(* Schneider Machine Expert - Basic project Run Hour, file version 1.7.0.0 *)
(* ProjectInformations: Name=New project *)

HARDWARE
  Cpu 0: TM221ME32TK
  EthernetConfiguration: NetworkName=M221, IpAllocationMode=FixedAddress, IpAddress=0.0.0.0, SubnetMask=0.0.0.0
  SerialLineConfiguration: Baud=Baud19200, Parity=ParityEven, DataBits=DataBits8, StopBits=StopBits1, PhysicalMedium=PhysicalMediumRs485, TransmissionMode=TransmissionModeModbusRtu, SlaveId=1, Addressing=SlaveAddressing
  MastTask: UsePeriodScanMode=false, PeriodScan=100
  FastTask: Period=255
  CpuBehavior: StartingMode=StartAsPreviousState, AutoSaveRamOnEeprom=true, WatchdogPeriod=250

SYMBOLS  (address, symbol, comment, settings)
  %TM1        "T1"  [Preset=5, Base=OneSecond]
  %TM2        "T2"  [Preset=5, Base=OneSecond]
  %TM3        [Base=OneSecond, IsRetentive=true]
  %TM4        [Base=OneSecond, IsRetentive=true]
  %I0.0       "Auto"
  %I0.1       "Manual"
  %I0.2       "Pompa 1"
  %I0.3       "Pompa 2"
  %Q0.0       "P1"
  %Q0.1       "P2"

POU New POU
  (* SectionNumber=1 *)

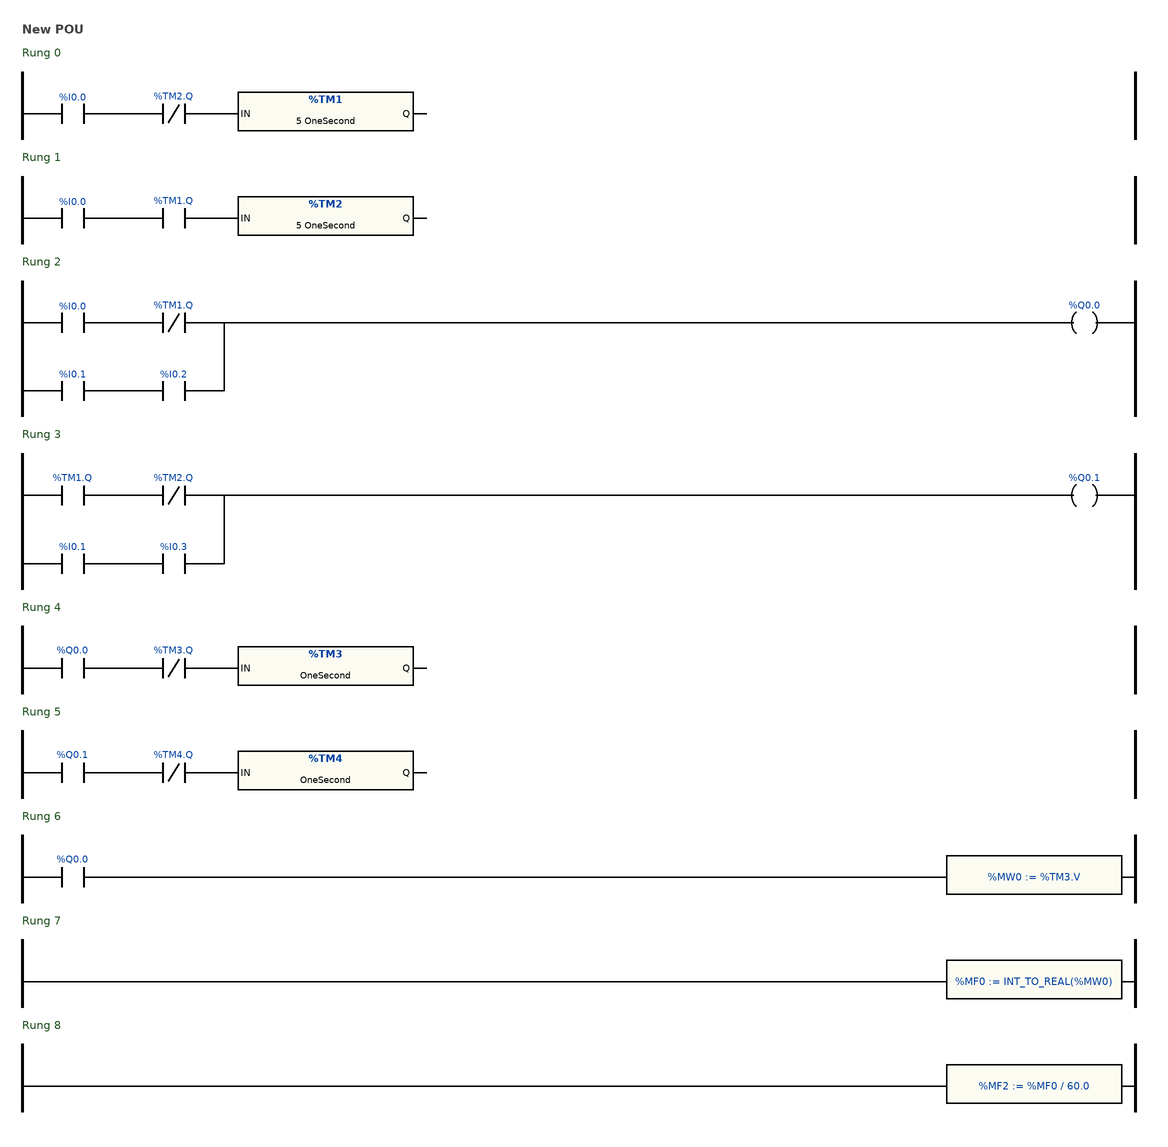

// Rung 0
  BLK %TM1
  LD %I0.0
  ANDN %TM2.Q
  IN
  END_BLK
  // as ST:
  //   %TM1(IN := %I0.0 AND NOT %TM2.Q);

// Rung 1
  BLK %TM2
  LD %I0.0
  AND %TM1.Q
  IN
  END_BLK
  // as ST:
  //   %TM2(IN := %I0.0 AND %TM1.Q);

// Rung 2
  LD %I0.0
  ANDN %TM1.Q
  OR( %I0.1
  AND %I0.2
  )
  ST %Q0.0
  // as ST:
  //   %Q0.0 := %I0.0 AND NOT %TM1.Q OR %I0.1 AND %I0.2;

// Rung 3
  LD %TM1.Q
  ANDN %TM2.Q
  OR( %I0.1
  AND %I0.3
  )
  ST %Q0.1
  // as ST:
  //   %Q0.1 := %TM1.Q AND NOT %TM2.Q OR %I0.1 AND %I0.3;

// Rung 4
  BLK %TM3
  LD %Q0.0
  ANDN %TM3.Q
  IN
  END_BLK
  // as ST:
  //   %TM3(IN := %Q0.0 AND NOT %TM3.Q);

// Rung 5
  BLK %TM4
  LD %Q0.1
  ANDN %TM4.Q
  IN
  END_BLK
  // as ST:
  //   %TM4(IN := %Q0.1 AND NOT %TM4.Q);

// Rung 6
  LD %Q0.0
  [ %MW0 := %TM3.V ]
  // as ST:
  //   IF %Q0.0 THEN %MW0 := %TM3.V; END_IF;

// Rung 7
  LD 1
  [ %MF0 := INT_TO_REAL ( %MW0 ) ]
  // as ST:
  //   %MF0 := INT_TO_REAL ( %MW0 );

// Rung 8
  LD 1
  [ %MF2 := %MF0 / 60.0 ]
  // as ST:
  //   %MF2 := %MF0  /  60.0;

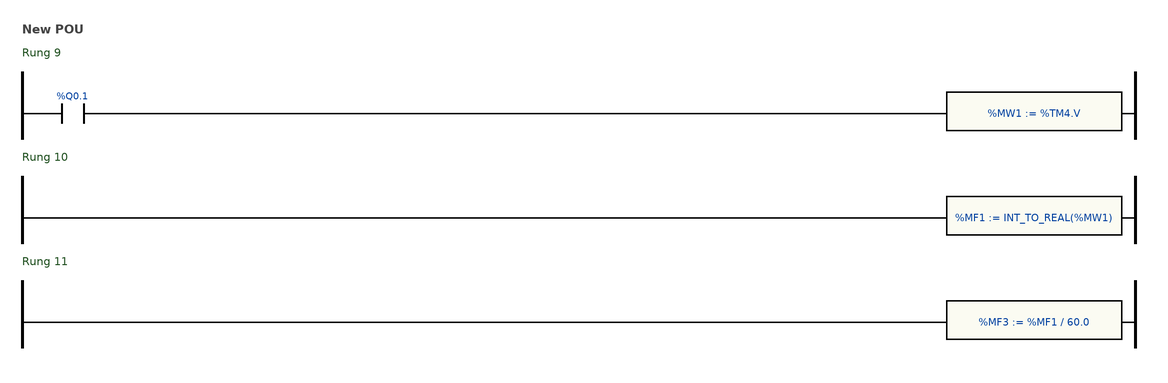

// Rung 9
  LD %Q0.1
  [ %MW1 := %TM4.V ]
  // as ST:
  //   IF %Q0.1 THEN %MW1 := %TM4.V; END_IF;

// Rung 10
  LD 1
  [ %MF1 := INT_TO_REAL ( %MW1 ) ]
  // as ST:
  //   %MF1 := INT_TO_REAL ( %MW1 );

// Rung 11
  LD 1
  [ %MF3 := %MF1 / 60.0 ]
  // as ST:
  //   %MF3 := %MF1  /  60.0;
